FUNCTION_BLOCK PassThrough_CTL
  (* Version 1.0, 2005-11-13, Goran Cengic, Chalmers *)
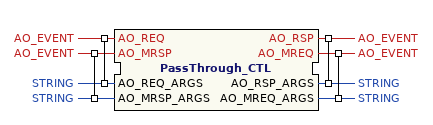
  EVENT_INPUT
    AO_REQ : AO_EVENT WITH AO_REQ_ARGS;
    AO_MRSP : AO_EVENT WITH AO_MRSP_ARGS;
  END_EVENT
  EVENT_OUTPUT
    AO_RSP : AO_EVENT WITH AO_RSP_ARGS;
    AO_MREQ : AO_EVENT WITH AO_MREQ_ARGS;
  END_EVENT
  VAR_INPUT
    AO_REQ_ARGS : STRING;
    AO_MRSP_ARGS : STRING;
  END_VAR
  VAR_OUTPUT
    AO_RSP_ARGS : STRING;
    AO_MREQ_ARGS : STRING;
  END_VAR
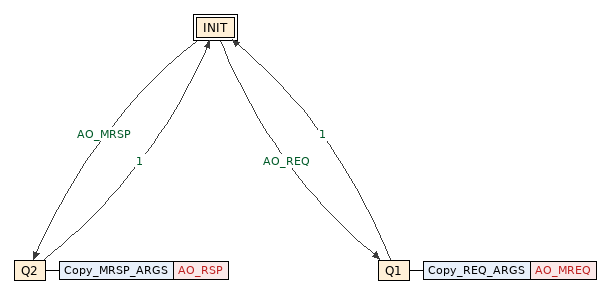
  EC_STATES
    INIT;
    Q1 : Copy_REQ_ARGS -> AO_MREQ;
    Q2 : Copy_MRSP_ARGS -> AO_RSP;
  END_STATES
  EC_TRANSITIONS
    INIT TO Q1 := AO_REQ;
    Q1 TO INIT := 1;
    INIT TO Q2 := AO_MRSP;
    Q2 TO INIT := 1;
  END_TRANSITIONS
  ALGORITHM Copy_REQ_ARGS IN Java:
AO_MREQ_ARGS = AO_REQ_ARGS;
  END_ALGORITHM
  ALGORITHM Copy_MRSP_ARGS IN Java:
AO_RSP_ARGS = AO_MRSP_ARGS;
  END_ALGORITHM
END_FUNCTION_BLOCK
